// TIA Portal V20 export
FUNCTION_BLOCK "CalculateCam_FeedingRoll"   // FB189, SCL
// stored: Access Published, MemoryReserve 100, SetENOAutomatically false
   VAR_INPUT
      targetCam : TO_Cam;
      excute { ExternalAccessible := 'False'; ExternalVisible := 'False'; ExternalWritable := 'False'} : Bool;
      cpm { ExternalAccessible := 'False'; ExternalVisible := 'False'; ExternalWritable := 'False'} : LReal;
      cellSize { ExternalAccessible := 'False'; ExternalVisible := 'False'; ExternalWritable := 'False'} : LReal;
   END_VAR
   VAR_OUTPUT
      done { ExternalAccessible := 'False'; ExternalVisible := 'False'; ExternalWritable := 'False'} : Bool;
      busy { ExternalAccessible := 'False'; ExternalVisible := 'False'; ExternalWritable := 'False'} : Bool;
      error { ExternalAccessible := 'False'; ExternalVisible := 'False'; ExternalWritable := 'False'} : Bool;
      errorID { ExternalAccessible := 'False'; ExternalVisible := 'False'; ExternalWritable := 'False'} : Word;
   END_VAR
   VAR
      instMCInterpolateCam { ExternalAccessible := 'False'; ExternalVisible := 'False'; ExternalWritable := 'False'} : MC_INTERPOLATECAM;
      statCmd { ExternalAccessible := 'False'; ExternalVisible := 'False'; ExternalWritable := 'False'; S7_SetPoint := 'True'} : DInt;
   END_VAR
   VAR_TEMP
      tempCycleTime : LReal;
      tempFeedingTime : LReal;
      tempT : LReal;
      tempCT : LReal;
      tempDT : LReal;
      tempL : LReal;
      tempR : LReal;
      tempCalPos : Array[1..15] of LReal;
      tempCalVel : Array[1..15] of LReal;
      tempCalAcc : Array[1..15] of LReal;
      tempJerk : Array[1..15] of LReal;
      tempAcc : Array[1..15] of LReal;
      tempVel : Array[1..15] of LReal;
      tempPos : Array[1..15] of LReal;
      tempTime : Array[1..15] of LReal;
      tempX : Array[1..15] of LReal;
      tempA0 : Array[1..50] of LReal;
      tempA1 : Array[1..50] of LReal;
      tempA2 : Array[1..50] of LReal;
      tempA3 : Array[1..50] of LReal;
      tempA4 : Array[1..50] of LReal;
      tempMax : Int;
   END_VAR
   VAR CONSTANT
      CC_IDLE : Int;
      CC_RESET : Int := 1;
      CC_CALCULATE : Int := 2;
      CC_INTERPOLATE : Int := 3;
      CC_DONE : Int := 4;
      CC_ERROR : Int := 99;
      BASIC_TIMEDIVE : LReal := 2.0;
      BASIC_FEEDERDIVE : LReal := 2.0;
      BASIC_ACCPART : Int := 3;
   END_VAR
BEGIN
   IF #instMCInterpolateCam.Error
   THEN
       #statCmd := #CC_ERROR;
       #errorID := #instMCInterpolateCam.ErrorId;
   END_IF;

   IF NOT #excute
   THEN
       #statCmd := #CC_IDLE;
   END_IF;
   REGION State machine
       CASE #statCmd
       OF
           #CC_IDLE:
               #errorID := 16#0;

               IF #excute
               THEN
                   #statCmd := #CC_RESET;
               END_IF;

           #CC_RESET:
               #targetCam.Segment[1].xmin := 0.0;
               #targetCam.Segment[2].xmin := 0.0;
               #targetCam.Segment[3].xmin := 0.0;
               #targetCam.Segment[4].xmin := 0.0;
               #targetCam.Segment[5].xmin := 0.0;
               #targetCam.Segment[6].xmin := 0.0;
               #targetCam.Segment[7].xmin := 0.0;
               #targetCam.Segment[8].xmin := 0.0;
               #targetCam.Segment[9].xmin := 0.0;
               #targetCam.Segment[10].xmin := 0.0;
               #targetCam.Segment[11].xmin := 0.0;
               #targetCam.Segment[12].xmin := 0.0;
               #targetCam.Segment[13].xmin := 0.0;
               #targetCam.Segment[14].xmin := 0.0;
               #targetCam.Segment[15].xmin := 0.0;
               #targetCam.Segment[16].xmin := 0.0;
               #targetCam.Segment[17].xmin := 0.0;
               #targetCam.Segment[18].xmin := 0.0;
               #targetCam.Segment[19].xmin := 0.0;
               #targetCam.Segment[20].xmin := 0.0;
               #targetCam.Segment[21].xmin := 0.0;
               #targetCam.Segment[22].xmin := 0.0;
               #targetCam.Segment[23].xmin := 0.0;
               #targetCam.Segment[24].xmin := 0.0;
               #targetCam.Segment[25].xmin := 0.0;
               #targetCam.Segment[26].xmin := 0.0;
               #targetCam.Segment[27].xmin := 0.0;
               #targetCam.Segment[28].xmin := 0.0;
               #targetCam.Segment[29].xmin := 0.0;
               #targetCam.Segment[30].xmin := 0.0;
               #targetCam.Segment[31].xmin := 0.0;
               #targetCam.Segment[32].xmin := 0.0;
               #targetCam.Segment[33].xmin := 0.0;
               #targetCam.Segment[34].xmin := 0.0;
               #targetCam.Segment[35].xmin := 0.0;
               #targetCam.Segment[36].xmin := 0.0;
               #targetCam.Segment[37].xmin := 0.0;
               #targetCam.Segment[38].xmin := 0.0;
               #targetCam.Segment[39].xmin := 0.0;
               #targetCam.Segment[40].xmin := 0.0;
               #targetCam.Segment[41].xmin := 0.0;
               #targetCam.Segment[42].xmin := 0.0;
               #targetCam.Segment[43].xmin := 0.0;
               #targetCam.Segment[44].xmin := 0.0;
               #targetCam.Segment[45].xmin := 0.0;
               #targetCam.Segment[46].xmin := 0.0;
               #targetCam.Segment[47].xmin := 0.0;
               #targetCam.Segment[48].xmin := 0.0;
               #targetCam.Segment[49].xmin := 0.0;
               #targetCam.Segment[50].xmin := 0.0;

               #targetCam.Segment[1].xmax := 0.0;
               #targetCam.Segment[2].xmax := 0.0;
               #targetCam.Segment[3].xmax := 0.0;
               #targetCam.Segment[4].xmax := 0.0;
               #targetCam.Segment[5].xmax := 0.0;
               #targetCam.Segment[6].xmax := 0.0;
               #targetCam.Segment[7].xmax := 0.0;
               #targetCam.Segment[8].xmax := 0.0;
               #targetCam.Segment[9].xmax := 0.0;
               #targetCam.Segment[10].xmax := 0.0;
               #targetCam.Segment[11].xmax := 0.0;
               #targetCam.Segment[12].xmax := 0.0;
               #targetCam.Segment[13].xmax := 0.0;
               #targetCam.Segment[14].xmax := 0.0;
               #targetCam.Segment[15].xmax := 0.0;
               #targetCam.Segment[16].xmax := 0.0;
               #targetCam.Segment[17].xmax := 0.0;
               #targetCam.Segment[18].xmax := 0.0;
               #targetCam.Segment[19].xmax := 0.0;
               #targetCam.Segment[20].xmax := 0.0;
               #targetCam.Segment[21].xmax := 0.0;
               #targetCam.Segment[22].xmax := 0.0;
               #targetCam.Segment[23].xmax := 0.0;
               #targetCam.Segment[24].xmax := 0.0;
               #targetCam.Segment[25].xmax := 0.0;
               #targetCam.Segment[26].xmax := 0.0;
               #targetCam.Segment[27].xmax := 0.0;
               #targetCam.Segment[28].xmax := 0.0;
               #targetCam.Segment[29].xmax := 0.0;
               #targetCam.Segment[30].xmax := 0.0;
               #targetCam.Segment[31].xmax := 0.0;
               #targetCam.Segment[32].xmax := 0.0;
               #targetCam.Segment[33].xmax := 0.0;
               #targetCam.Segment[34].xmax := 0.0;
               #targetCam.Segment[35].xmax := 0.0;
               #targetCam.Segment[36].xmax := 0.0;
               #targetCam.Segment[37].xmax := 0.0;
               #targetCam.Segment[38].xmax := 0.0;
               #targetCam.Segment[39].xmax := 0.0;
               #targetCam.Segment[40].xmax := 0.0;
               #targetCam.Segment[41].xmax := 0.0;
               #targetCam.Segment[42].xmax := 0.0;
               #targetCam.Segment[43].xmax := 0.0;
               #targetCam.Segment[44].xmax := 0.0;
               #targetCam.Segment[45].xmax := 0.0;
               #targetCam.Segment[46].xmax := 0.0;
               #targetCam.Segment[47].xmax := 0.0;
               #targetCam.Segment[48].xmax := 0.0;
               #targetCam.Segment[49].xmax := 0.0;
               #targetCam.Segment[50].xmax := 0.0;

               #targetCam.Segment[1].a0 := 0.0;
               #targetCam.Segment[2].a0 := 0.0;
               #targetCam.Segment[3].a0 := 0.0;
               #targetCam.Segment[4].a0 := 0.0;
               #targetCam.Segment[5].a0 := 0.0;
               #targetCam.Segment[6].a0 := 0.0;
               #targetCam.Segment[7].a0 := 0.0;
               #targetCam.Segment[8].a0 := 0.0;
               #targetCam.Segment[9].a0 := 0.0;
               #targetCam.Segment[10].a0 := 0.0;
               #targetCam.Segment[11].a0 := 0.0;
               #targetCam.Segment[12].a0 := 0.0;
               #targetCam.Segment[13].a0 := 0.0;
               #targetCam.Segment[14].a0 := 0.0;
               #targetCam.Segment[15].a0 := 0.0;
               #targetCam.Segment[16].a0 := 0.0;
               #targetCam.Segment[17].a0 := 0.0;
               #targetCam.Segment[18].a0 := 0.0;
               #targetCam.Segment[19].a0 := 0.0;
               #targetCam.Segment[20].a0 := 0.0;
               #targetCam.Segment[21].a0 := 0.0;
               #targetCam.Segment[22].a0 := 0.0;
               #targetCam.Segment[23].a0 := 0.0;
               #targetCam.Segment[24].a0 := 0.0;
               #targetCam.Segment[25].a0 := 0.0;
               #targetCam.Segment[26].a0 := 0.0;
               #targetCam.Segment[27].a0 := 0.0;
               #targetCam.Segment[28].a0 := 0.0;
               #targetCam.Segment[29].a0 := 0.0;
               #targetCam.Segment[30].a0 := 0.0;
               #targetCam.Segment[31].a0 := 0.0;
               #targetCam.Segment[32].a0 := 0.0;
               #targetCam.Segment[33].a0 := 0.0;
               #targetCam.Segment[34].a0 := 0.0;
               #targetCam.Segment[35].a0 := 0.0;
               #targetCam.Segment[36].a0 := 0.0;
               #targetCam.Segment[37].a0 := 0.0;
               #targetCam.Segment[38].a0 := 0.0;
               #targetCam.Segment[39].a0 := 0.0;
               #targetCam.Segment[40].a0 := 0.0;
               #targetCam.Segment[41].a0 := 0.0;
               #targetCam.Segment[42].a0 := 0.0;
               #targetCam.Segment[43].a0 := 0.0;
               #targetCam.Segment[44].a0 := 0.0;
               #targetCam.Segment[45].a0 := 0.0;
               #targetCam.Segment[46].a0 := 0.0;
               #targetCam.Segment[47].a0 := 0.0;
               #targetCam.Segment[48].a0 := 0.0;
               #targetCam.Segment[49].a0 := 0.0;
               #targetCam.Segment[50].a0 := 0.0;

               #targetCam.Segment[1].a1 := 0.0;
               #targetCam.Segment[2].a1 := 0.0;
               #targetCam.Segment[3].a1 := 0.0;
               #targetCam.Segment[4].a1 := 0.0;
               #targetCam.Segment[5].a1 := 0.0;
               #targetCam.Segment[6].a1 := 0.0;
               #targetCam.Segment[7].a1 := 0.0;
               #targetCam.Segment[8].a1 := 0.0;
               #targetCam.Segment[9].a1 := 0.0;
               #targetCam.Segment[10].a1 := 0.0;
               #targetCam.Segment[11].a1 := 0.0;
               #targetCam.Segment[12].a1 := 0.0;
               #targetCam.Segment[13].a1 := 0.0;
               #targetCam.Segment[14].a1 := 0.0;
               #targetCam.Segment[15].a1 := 0.0;
               #targetCam.Segment[16].a1 := 0.0;
               #targetCam.Segment[17].a1 := 0.0;
               #targetCam.Segment[18].a1 := 0.0;
               #targetCam.Segment[19].a1 := 0.0;
               #targetCam.Segment[20].a1 := 0.0;
               #targetCam.Segment[21].a1 := 0.0;
               #targetCam.Segment[22].a1 := 0.0;
               #targetCam.Segment[23].a1 := 0.0;
               #targetCam.Segment[24].a1 := 0.0;
               #targetCam.Segment[25].a1 := 0.0;
               #targetCam.Segment[26].a1 := 0.0;
               #targetCam.Segment[27].a1 := 0.0;
               #targetCam.Segment[28].a1 := 0.0;
               #targetCam.Segment[29].a1 := 0.0;
               #targetCam.Segment[30].a1 := 0.0;
               #targetCam.Segment[31].a1 := 0.0;
               #targetCam.Segment[32].a1 := 0.0;
               #targetCam.Segment[33].a1 := 0.0;
               #targetCam.Segment[34].a1 := 0.0;
               #targetCam.Segment[35].a1 := 0.0;
               #targetCam.Segment[36].a1 := 0.0;
               #targetCam.Segment[37].a1 := 0.0;
               #targetCam.Segment[38].a1 := 0.0;
               #targetCam.Segment[39].a1 := 0.0;
               #targetCam.Segment[40].a1 := 0.0;
               #targetCam.Segment[41].a1 := 0.0;
               #targetCam.Segment[42].a1 := 0.0;
               #targetCam.Segment[43].a1 := 0.0;
               #targetCam.Segment[44].a1 := 0.0;
               #targetCam.Segment[45].a1 := 0.0;
               #targetCam.Segment[46].a1 := 0.0;
               #targetCam.Segment[47].a1 := 0.0;
               #targetCam.Segment[48].a1 := 0.0;
               #targetCam.Segment[49].a1 := 0.0;
               #targetCam.Segment[50].a1 := 0.0;

               #targetCam.Segment[1].a2 := 0.0;
               #targetCam.Segment[2].a2 := 0.0;
               #targetCam.Segment[3].a2 := 0.0;
               #targetCam.Segment[4].a2 := 0.0;
               #targetCam.Segment[5].a2 := 0.0;
               #targetCam.Segment[6].a2 := 0.0;
               #targetCam.Segment[7].a2 := 0.0;
               #targetCam.Segment[8].a2 := 0.0;
               #targetCam.Segment[9].a2 := 0.0;
               #targetCam.Segment[10].a2 := 0.0;
               #targetCam.Segment[11].a2 := 0.0;
               #targetCam.Segment[12].a2 := 0.0;
               #targetCam.Segment[13].a2 := 0.0;
               #targetCam.Segment[14].a2 := 0.0;
               #targetCam.Segment[15].a2 := 0.0;
               #targetCam.Segment[16].a2 := 0.0;
               #targetCam.Segment[17].a2 := 0.0;
               #targetCam.Segment[18].a2 := 0.0;
               #targetCam.Segment[19].a2 := 0.0;
               #targetCam.Segment[20].a2 := 0.0;
               #targetCam.Segment[21].a2 := 0.0;
               #targetCam.Segment[22].a2 := 0.0;
               #targetCam.Segment[23].a2 := 0.0;
               #targetCam.Segment[24].a2 := 0.0;
               #targetCam.Segment[25].a2 := 0.0;
               #targetCam.Segment[26].a2 := 0.0;
               #targetCam.Segment[27].a2 := 0.0;
               #targetCam.Segment[28].a2 := 0.0;
               #targetCam.Segment[29].a2 := 0.0;
               #targetCam.Segment[30].a2 := 0.0;
               #targetCam.Segment[31].a2 := 0.0;
               #targetCam.Segment[32].a2 := 0.0;
               #targetCam.Segment[33].a2 := 0.0;
               #targetCam.Segment[34].a2 := 0.0;
               #targetCam.Segment[35].a2 := 0.0;
               #targetCam.Segment[36].a2 := 0.0;
               #targetCam.Segment[37].a2 := 0.0;
               #targetCam.Segment[38].a2 := 0.0;
               #targetCam.Segment[39].a2 := 0.0;
               #targetCam.Segment[40].a2 := 0.0;
               #targetCam.Segment[41].a2 := 0.0;
               #targetCam.Segment[42].a2 := 0.0;
               #targetCam.Segment[43].a2 := 0.0;
               #targetCam.Segment[44].a2 := 0.0;
               #targetCam.Segment[45].a2 := 0.0;
               #targetCam.Segment[46].a2 := 0.0;
               #targetCam.Segment[47].a2 := 0.0;
               #targetCam.Segment[48].a2 := 0.0;
               #targetCam.Segment[49].a2 := 0.0;
               #targetCam.Segment[50].a2 := 0.0;

               #targetCam.Segment[1].a3 := 0.0;
               #targetCam.Segment[2].a3 := 0.0;
               #targetCam.Segment[3].a3 := 0.0;
               #targetCam.Segment[4].a3 := 0.0;
               #targetCam.Segment[5].a3 := 0.0;
               #targetCam.Segment[6].a3 := 0.0;
               #targetCam.Segment[7].a3 := 0.0;
               #targetCam.Segment[8].a3 := 0.0;
               #targetCam.Segment[9].a3 := 0.0;
               #targetCam.Segment[10].a3 := 0.0;
               #targetCam.Segment[11].a3 := 0.0;
               #targetCam.Segment[12].a3 := 0.0;
               #targetCam.Segment[13].a3 := 0.0;
               #targetCam.Segment[14].a3 := 0.0;
               #targetCam.Segment[15].a3 := 0.0;
               #targetCam.Segment[16].a3 := 0.0;
               #targetCam.Segment[17].a3 := 0.0;
               #targetCam.Segment[18].a3 := 0.0;
               #targetCam.Segment[19].a3 := 0.0;
               #targetCam.Segment[20].a3 := 0.0;
               #targetCam.Segment[21].a3 := 0.0;
               #targetCam.Segment[22].a3 := 0.0;
               #targetCam.Segment[23].a3 := 0.0;
               #targetCam.Segment[24].a3 := 0.0;
               #targetCam.Segment[25].a3 := 0.0;
               #targetCam.Segment[26].a3 := 0.0;
               #targetCam.Segment[27].a3 := 0.0;
               #targetCam.Segment[28].a3 := 0.0;
               #targetCam.Segment[29].a3 := 0.0;
               #targetCam.Segment[30].a3 := 0.0;
               #targetCam.Segment[31].a3 := 0.0;
               #targetCam.Segment[32].a3 := 0.0;
               #targetCam.Segment[33].a3 := 0.0;
               #targetCam.Segment[34].a3 := 0.0;
               #targetCam.Segment[35].a3 := 0.0;
               #targetCam.Segment[36].a3 := 0.0;
               #targetCam.Segment[37].a3 := 0.0;
               #targetCam.Segment[38].a3 := 0.0;
               #targetCam.Segment[39].a3 := 0.0;
               #targetCam.Segment[40].a3 := 0.0;
               #targetCam.Segment[41].a3 := 0.0;
               #targetCam.Segment[42].a3 := 0.0;
               #targetCam.Segment[43].a3 := 0.0;
               #targetCam.Segment[44].a3 := 0.0;
               #targetCam.Segment[45].a3 := 0.0;
               #targetCam.Segment[46].a3 := 0.0;
               #targetCam.Segment[47].a3 := 0.0;
               #targetCam.Segment[48].a3 := 0.0;
               #targetCam.Segment[49].a3 := 0.0;
               #targetCam.Segment[50].a3 := 0.0;

               #targetCam.Segment[1].a4 := 0.0;
               #targetCam.Segment[2].a4 := 0.0;
               #targetCam.Segment[3].a4 := 0.0;
               #targetCam.Segment[4].a4 := 0.0;
               #targetCam.Segment[5].a4 := 0.0;
               #targetCam.Segment[6].a4 := 0.0;
               #targetCam.Segment[7].a4 := 0.0;
               #targetCam.Segment[8].a4 := 0.0;
               #targetCam.Segment[9].a4 := 0.0;
               #targetCam.Segment[10].a4 := 0.0;
               #targetCam.Segment[11].a4 := 0.0;
               #targetCam.Segment[12].a4 := 0.0;
               #targetCam.Segment[13].a4 := 0.0;
               #targetCam.Segment[14].a4 := 0.0;
               #targetCam.Segment[15].a4 := 0.0;
               #targetCam.Segment[16].a4 := 0.0;
               #targetCam.Segment[17].a4 := 0.0;
               #targetCam.Segment[18].a4 := 0.0;
               #targetCam.Segment[19].a4 := 0.0;
               #targetCam.Segment[20].a4 := 0.0;
               #targetCam.Segment[21].a4 := 0.0;
               #targetCam.Segment[22].a4 := 0.0;
               #targetCam.Segment[23].a4 := 0.0;
               #targetCam.Segment[24].a4 := 0.0;
               #targetCam.Segment[25].a4 := 0.0;
               #targetCam.Segment[26].a4 := 0.0;
               #targetCam.Segment[27].a4 := 0.0;
               #targetCam.Segment[28].a4 := 0.0;
               #targetCam.Segment[29].a4 := 0.0;
               #targetCam.Segment[30].a4 := 0.0;
               #targetCam.Segment[31].a4 := 0.0;
               #targetCam.Segment[32].a4 := 0.0;
               #targetCam.Segment[33].a4 := 0.0;
               #targetCam.Segment[34].a4 := 0.0;
               #targetCam.Segment[35].a4 := 0.0;
               #targetCam.Segment[36].a4 := 0.0;
               #targetCam.Segment[37].a4 := 0.0;
               #targetCam.Segment[38].a4 := 0.0;
               #targetCam.Segment[39].a4 := 0.0;
               #targetCam.Segment[40].a4 := 0.0;
               #targetCam.Segment[41].a4 := 0.0;
               #targetCam.Segment[42].a4 := 0.0;
               #targetCam.Segment[43].a4 := 0.0;
               #targetCam.Segment[44].a4 := 0.0;
               #targetCam.Segment[45].a4 := 0.0;
               #targetCam.Segment[46].a4 := 0.0;
               #targetCam.Segment[47].a4 := 0.0;
               #targetCam.Segment[48].a4 := 0.0;
               #targetCam.Segment[49].a4 := 0.0;
               #targetCam.Segment[50].a4 := 0.0;

               #targetCam.Segment[1].a5 := 0.0;
               #targetCam.Segment[2].a5 := 0.0;
               #targetCam.Segment[3].a5 := 0.0;
               #targetCam.Segment[4].a5 := 0.0;
               #targetCam.Segment[5].a5 := 0.0;
               #targetCam.Segment[6].a5 := 0.0;
               #targetCam.Segment[7].a5 := 0.0;
               #targetCam.Segment[8].a5 := 0.0;
               #targetCam.Segment[9].a5 := 0.0;
               #targetCam.Segment[10].a5 := 0.0;
               #targetCam.Segment[11].a5 := 0.0;
               #targetCam.Segment[12].a5 := 0.0;
               #targetCam.Segment[13].a5 := 0.0;
               #targetCam.Segment[14].a5 := 0.0;
               #targetCam.Segment[15].a5 := 0.0;
               #targetCam.Segment[16].a5 := 0.0;
               #targetCam.Segment[17].a5 := 0.0;
               #targetCam.Segment[18].a5 := 0.0;
               #targetCam.Segment[19].a5 := 0.0;
               #targetCam.Segment[20].a5 := 0.0;
               #targetCam.Segment[21].a5 := 0.0;
               #targetCam.Segment[22].a5 := 0.0;
               #targetCam.Segment[23].a5 := 0.0;
               #targetCam.Segment[24].a5 := 0.0;
               #targetCam.Segment[25].a5 := 0.0;
               #targetCam.Segment[26].a5 := 0.0;
               #targetCam.Segment[27].a5 := 0.0;
               #targetCam.Segment[28].a5 := 0.0;
               #targetCam.Segment[29].a5 := 0.0;
               #targetCam.Segment[30].a5 := 0.0;
               #targetCam.Segment[31].a5 := 0.0;
               #targetCam.Segment[32].a5 := 0.0;
               #targetCam.Segment[33].a5 := 0.0;
               #targetCam.Segment[34].a5 := 0.0;
               #targetCam.Segment[35].a5 := 0.0;
               #targetCam.Segment[36].a5 := 0.0;
               #targetCam.Segment[37].a5 := 0.0;
               #targetCam.Segment[38].a5 := 0.0;
               #targetCam.Segment[39].a5 := 0.0;
               #targetCam.Segment[40].a5 := 0.0;
               #targetCam.Segment[41].a5 := 0.0;
               #targetCam.Segment[42].a5 := 0.0;
               #targetCam.Segment[43].a5 := 0.0;
               #targetCam.Segment[44].a5 := 0.0;
               #targetCam.Segment[45].a5 := 0.0;
               #targetCam.Segment[46].a5 := 0.0;
               #targetCam.Segment[47].a5 := 0.0;
               #targetCam.Segment[48].a5 := 0.0;
               #targetCam.Segment[49].a5 := 0.0;
               #targetCam.Segment[50].a5 := 0.0;

               #targetCam.Segment[1].a6 := 0.0;
               #targetCam.Segment[2].a6 := 0.0;
               #targetCam.Segment[3].a6 := 0.0;
               #targetCam.Segment[4].a6 := 0.0;
               #targetCam.Segment[5].a6 := 0.0;
               #targetCam.Segment[6].a6 := 0.0;
               #targetCam.Segment[7].a6 := 0.0;
               #targetCam.Segment[8].a6 := 0.0;
               #targetCam.Segment[9].a6 := 0.0;
               #targetCam.Segment[10].a6 := 0.0;
               #targetCam.Segment[11].a6 := 0.0;
               #targetCam.Segment[12].a6 := 0.0;
               #targetCam.Segment[13].a6 := 0.0;
               #targetCam.Segment[14].a6 := 0.0;
               #targetCam.Segment[15].a6 := 0.0;
               #targetCam.Segment[16].a6 := 0.0;
               #targetCam.Segment[17].a6 := 0.0;
               #targetCam.Segment[18].a6 := 0.0;
               #targetCam.Segment[19].a6 := 0.0;
               #targetCam.Segment[20].a6 := 0.0;
               #targetCam.Segment[21].a6 := 0.0;
               #targetCam.Segment[22].a6 := 0.0;
               #targetCam.Segment[23].a6 := 0.0;
               #targetCam.Segment[24].a6 := 0.0;
               #targetCam.Segment[25].a6 := 0.0;
               #targetCam.Segment[26].a6 := 0.0;
               #targetCam.Segment[27].a6 := 0.0;
               #targetCam.Segment[28].a6 := 0.0;
               #targetCam.Segment[29].a6 := 0.0;
               #targetCam.Segment[30].a6 := 0.0;
               #targetCam.Segment[31].a6 := 0.0;
               #targetCam.Segment[32].a6 := 0.0;
               #targetCam.Segment[33].a6 := 0.0;
               #targetCam.Segment[34].a6 := 0.0;
               #targetCam.Segment[35].a6 := 0.0;
               #targetCam.Segment[36].a6 := 0.0;
               #targetCam.Segment[37].a6 := 0.0;
               #targetCam.Segment[38].a6 := 0.0;
               #targetCam.Segment[39].a6 := 0.0;
               #targetCam.Segment[40].a6 := 0.0;
               #targetCam.Segment[41].a6 := 0.0;
               #targetCam.Segment[42].a6 := 0.0;
               #targetCam.Segment[43].a6 := 0.0;
               #targetCam.Segment[44].a6 := 0.0;
               #targetCam.Segment[45].a6 := 0.0;
               #targetCam.Segment[46].a6 := 0.0;
               #targetCam.Segment[47].a6 := 0.0;
               #targetCam.Segment[48].a6 := 0.0;
               #targetCam.Segment[49].a6 := 0.0;
               #targetCam.Segment[50].a6 := 0.0;

               #targetCam.Segment[1].sineAmplitude := 0.0;
               #targetCam.Segment[2].sineAmplitude := 0.0;
               #targetCam.Segment[3].sineAmplitude := 0.0;
               #targetCam.Segment[4].sineAmplitude := 0.0;
               #targetCam.Segment[5].sineAmplitude := 0.0;
               #targetCam.Segment[6].sineAmplitude := 0.0;
               #targetCam.Segment[7].sineAmplitude := 0.0;
               #targetCam.Segment[8].sineAmplitude := 0.0;
               #targetCam.Segment[9].sineAmplitude := 0.0;
               #targetCam.Segment[10].sineAmplitude := 0.0;
               #targetCam.Segment[11].sineAmplitude := 0.0;
               #targetCam.Segment[12].sineAmplitude := 0.0;
               #targetCam.Segment[13].sineAmplitude := 0.0;
               #targetCam.Segment[14].sineAmplitude := 0.0;
               #targetCam.Segment[15].sineAmplitude := 0.0;
               #targetCam.Segment[16].sineAmplitude := 0.0;
               #targetCam.Segment[17].sineAmplitude := 0.0;
               #targetCam.Segment[18].sineAmplitude := 0.0;
               #targetCam.Segment[19].sineAmplitude := 0.0;
               #targetCam.Segment[20].sineAmplitude := 0.0;
               #targetCam.Segment[21].sineAmplitude := 0.0;
               #targetCam.Segment[22].sineAmplitude := 0.0;
               #targetCam.Segment[23].sineAmplitude := 0.0;
               #targetCam.Segment[24].sineAmplitude := 0.0;
               #targetCam.Segment[25].sineAmplitude := 0.0;
               #targetCam.Segment[26].sineAmplitude := 0.0;
               #targetCam.Segment[27].sineAmplitude := 0.0;
               #targetCam.Segment[28].sineAmplitude := 0.0;
               #targetCam.Segment[29].sineAmplitude := 0.0;
               #targetCam.Segment[30].sineAmplitude := 0.0;
               #targetCam.Segment[31].sineAmplitude := 0.0;
               #targetCam.Segment[32].sineAmplitude := 0.0;
               #targetCam.Segment[33].sineAmplitude := 0.0;
               #targetCam.Segment[34].sineAmplitude := 0.0;
               #targetCam.Segment[35].sineAmplitude := 0.0;
               #targetCam.Segment[36].sineAmplitude := 0.0;
               #targetCam.Segment[37].sineAmplitude := 0.0;
               #targetCam.Segment[38].sineAmplitude := 0.0;
               #targetCam.Segment[39].sineAmplitude := 0.0;
               #targetCam.Segment[40].sineAmplitude := 0.0;
               #targetCam.Segment[41].sineAmplitude := 0.0;
               #targetCam.Segment[42].sineAmplitude := 0.0;
               #targetCam.Segment[43].sineAmplitude := 0.0;
               #targetCam.Segment[44].sineAmplitude := 0.0;
               #targetCam.Segment[45].sineAmplitude := 0.0;
               #targetCam.Segment[46].sineAmplitude := 0.0;
               #targetCam.Segment[47].sineAmplitude := 0.0;
               #targetCam.Segment[48].sineAmplitude := 0.0;
               #targetCam.Segment[49].sineAmplitude := 0.0;
               #targetCam.Segment[50].sineAmplitude := 0.0;

               #targetCam.Segment[1].sinePeriod := 0.0;
               #targetCam.Segment[2].sinePeriod := 0.0;
               #targetCam.Segment[3].sinePeriod := 0.0;
               #targetCam.Segment[4].sinePeriod := 0.0;
               #targetCam.Segment[5].sinePeriod := 0.0;
               #targetCam.Segment[6].sinePeriod := 0.0;
               #targetCam.Segment[7].sinePeriod := 0.0;
               #targetCam.Segment[8].sinePeriod := 0.0;
               #targetCam.Segment[9].sinePeriod := 0.0;
               #targetCam.Segment[10].sinePeriod := 0.0;
               #targetCam.Segment[11].sinePeriod := 0.0;
               #targetCam.Segment[12].sinePeriod := 0.0;
               #targetCam.Segment[13].sinePeriod := 0.0;
               #targetCam.Segment[14].sinePeriod := 0.0;
               #targetCam.Segment[15].sinePeriod := 0.0;
               #targetCam.Segment[16].sinePeriod := 0.0;
               #targetCam.Segment[17].sinePeriod := 0.0;
               #targetCam.Segment[18].sinePeriod := 0.0;
               #targetCam.Segment[19].sinePeriod := 0.0;
               #targetCam.Segment[20].sinePeriod := 0.0;
               #targetCam.Segment[21].sinePeriod := 0.0;
               #targetCam.Segment[22].sinePeriod := 0.0;
               #targetCam.Segment[23].sinePeriod := 0.0;
               #targetCam.Segment[24].sinePeriod := 0.0;
               #targetCam.Segment[25].sinePeriod := 0.0;
               #targetCam.Segment[26].sinePeriod := 0.0;
               #targetCam.Segment[27].sinePeriod := 0.0;
               #targetCam.Segment[28].sinePeriod := 0.0;
               #targetCam.Segment[29].sinePeriod := 0.0;
               #targetCam.Segment[30].sinePeriod := 0.0;
               #targetCam.Segment[31].sinePeriod := 0.0;
               #targetCam.Segment[32].sinePeriod := 0.0;
               #targetCam.Segment[33].sinePeriod := 0.0;
               #targetCam.Segment[34].sinePeriod := 0.0;
               #targetCam.Segment[35].sinePeriod := 0.0;
               #targetCam.Segment[36].sinePeriod := 0.0;
               #targetCam.Segment[37].sinePeriod := 0.0;
               #targetCam.Segment[38].sinePeriod := 0.0;
               #targetCam.Segment[39].sinePeriod := 0.0;
               #targetCam.Segment[40].sinePeriod := 0.0;
               #targetCam.Segment[41].sinePeriod := 0.0;
               #targetCam.Segment[42].sinePeriod := 0.0;
               #targetCam.Segment[43].sinePeriod := 0.0;
               #targetCam.Segment[44].sinePeriod := 0.0;
               #targetCam.Segment[45].sinePeriod := 0.0;
               #targetCam.Segment[46].sinePeriod := 0.0;
               #targetCam.Segment[47].sinePeriod := 0.0;
               #targetCam.Segment[48].sinePeriod := 0.0;
               #targetCam.Segment[49].sinePeriod := 0.0;
               #targetCam.Segment[50].sinePeriod := 0.0;

               #targetCam.Segment[1].sinePhase := 0.0;
               #targetCam.Segment[2].sinePhase := 0.0;
               #targetCam.Segment[3].sinePhase := 0.0;
               #targetCam.Segment[4].sinePhase := 0.0;
               #targetCam.Segment[5].sinePhase := 0.0;
               #targetCam.Segment[6].sinePhase := 0.0;
               #targetCam.Segment[7].sinePhase := 0.0;
               #targetCam.Segment[8].sinePhase := 0.0;
               #targetCam.Segment[9].sinePhase := 0.0;
               #targetCam.Segment[10].sinePhase := 0.0;
               #targetCam.Segment[11].sinePhase := 0.0;
               #targetCam.Segment[12].sinePhase := 0.0;
               #targetCam.Segment[13].sinePhase := 0.0;
               #targetCam.Segment[14].sinePhase := 0.0;
               #targetCam.Segment[15].sinePhase := 0.0;
               #targetCam.Segment[16].sinePhase := 0.0;
               #targetCam.Segment[17].sinePhase := 0.0;
               #targetCam.Segment[18].sinePhase := 0.0;
               #targetCam.Segment[19].sinePhase := 0.0;
               #targetCam.Segment[20].sinePhase := 0.0;
               #targetCam.Segment[21].sinePhase := 0.0;
               #targetCam.Segment[22].sinePhase := 0.0;
               #targetCam.Segment[23].sinePhase := 0.0;
               #targetCam.Segment[24].sinePhase := 0.0;
               #targetCam.Segment[25].sinePhase := 0.0;
               #targetCam.Segment[26].sinePhase := 0.0;
               #targetCam.Segment[27].sinePhase := 0.0;
               #targetCam.Segment[28].sinePhase := 0.0;
               #targetCam.Segment[29].sinePhase := 0.0;
               #targetCam.Segment[30].sinePhase := 0.0;
               #targetCam.Segment[31].sinePhase := 0.0;
               #targetCam.Segment[32].sinePhase := 0.0;
               #targetCam.Segment[33].sinePhase := 0.0;
               #targetCam.Segment[34].sinePhase := 0.0;
               #targetCam.Segment[35].sinePhase := 0.0;
               #targetCam.Segment[36].sinePhase := 0.0;
               #targetCam.Segment[37].sinePhase := 0.0;
               #targetCam.Segment[38].sinePhase := 0.0;
               #targetCam.Segment[39].sinePhase := 0.0;
               #targetCam.Segment[40].sinePhase := 0.0;
               #targetCam.Segment[41].sinePhase := 0.0;
               #targetCam.Segment[42].sinePhase := 0.0;
               #targetCam.Segment[43].sinePhase := 0.0;
               #targetCam.Segment[44].sinePhase := 0.0;
               #targetCam.Segment[45].sinePhase := 0.0;
               #targetCam.Segment[46].sinePhase := 0.0;
               #targetCam.Segment[47].sinePhase := 0.0;
               #targetCam.Segment[48].sinePhase := 0.0;
               #targetCam.Segment[49].sinePhase := 0.0;
               #targetCam.Segment[50].sinePhase := 0.0;

               #targetCam.ValidSegment[1] := FALSE;
               #targetCam.ValidSegment[2] := FALSE;
               #targetCam.ValidSegment[3] := FALSE;
               #targetCam.ValidSegment[4] := FALSE;
               #targetCam.ValidSegment[5] := FALSE;
               #targetCam.ValidSegment[6] := FALSE;
               #targetCam.ValidSegment[7] := FALSE;
               #targetCam.ValidSegment[8] := FALSE;
               #targetCam.ValidSegment[9] := FALSE;
               #targetCam.ValidSegment[10] := FALSE;
               #targetCam.ValidSegment[11] := FALSE;
               #targetCam.ValidSegment[12] := FALSE;
               #targetCam.ValidSegment[13] := FALSE;
               #targetCam.ValidSegment[14] := FALSE;
               #targetCam.ValidSegment[15] := FALSE;
               #targetCam.ValidSegment[16] := FALSE;
               #targetCam.ValidSegment[17] := FALSE;
               #targetCam.ValidSegment[18] := FALSE;
               #targetCam.ValidSegment[19] := FALSE;
               #targetCam.ValidSegment[20] := FALSE;
               #targetCam.ValidSegment[21] := FALSE;
               #targetCam.ValidSegment[22] := FALSE;
               #targetCam.ValidSegment[23] := FALSE;
               #targetCam.ValidSegment[24] := FALSE;
               #targetCam.ValidSegment[25] := FALSE;
               #targetCam.ValidSegment[26] := FALSE;
               #targetCam.ValidSegment[27] := FALSE;
               #targetCam.ValidSegment[28] := FALSE;
               #targetCam.ValidSegment[29] := FALSE;
               #targetCam.ValidSegment[30] := FALSE;
               #targetCam.ValidSegment[31] := FALSE;
               #targetCam.ValidSegment[32] := FALSE;
               #targetCam.ValidSegment[33] := FALSE;
               #targetCam.ValidSegment[34] := FALSE;
               #targetCam.ValidSegment[35] := FALSE;
               #targetCam.ValidSegment[36] := FALSE;
               #targetCam.ValidSegment[37] := FALSE;
               #targetCam.ValidSegment[38] := FALSE;
               #targetCam.ValidSegment[39] := FALSE;
               #targetCam.ValidSegment[40] := FALSE;
               #targetCam.ValidSegment[41] := FALSE;
               #targetCam.ValidSegment[42] := FALSE;
               #targetCam.ValidSegment[43] := FALSE;
               #targetCam.ValidSegment[44] := FALSE;
               #targetCam.ValidSegment[45] := FALSE;
               #targetCam.ValidSegment[46] := FALSE;
               #targetCam.ValidSegment[47] := FALSE;
               #targetCam.ValidSegment[48] := FALSE;
               #targetCam.ValidSegment[49] := FALSE;
               #targetCam.ValidSegment[50] := FALSE;

               #statCmd := #CC_CALCULATE;

           #CC_CALCULATE:

               // Calculate Value
               #tempCycleTime := 60000.0 / #cpm;
               // CycleTime Calculate
               #tempFeedingTime := #tempCycleTime / #BASIC_TIMEDIVE;
               #tempT := #tempFeedingTime / 2.0;
               // TimePart Calculate Time / 3
               #tempL := #cpm * #cellSize / 60.0;
               #tempR := #cellSize / #tempT * 1000.0;
               // VelocityPart Calculate
               // 
               #tempTime[1] := 0.0;
               #tempTime[2] := #tempL * #tempT / 1000.0;
               #tempTime[3] := #tempL * #tempT / 1000.0;
               #tempTime[4] := 0.0;
               // Calculate Time

               #tempPos[1] := 0.0;
               #tempPos[2] := #tempR * #tempT / 1000.0 / 2.0;
               #tempPos[3] := #tempR * #tempT / 1000.0 / 2.0;
               #tempPos[4] := 0.0;
               // Calculate Pos

               #tempVel[1] := 0.0;
               #tempVel[2] := 2.0 * #tempPos[2] / #tempTime[2];
               #tempVel[3] := 2.0 * #tempPos[3] / #tempTime[3];
               #tempVel[4] := 0.0;

               // Calculate New Vel

               #tempAcc[1] := 0.0;
               #tempAcc[2] := 2.0 * #tempVel[2] / #tempTime[2];
               #tempAcc[3] := - 2.0 * #tempVel[3] / #tempTime[3];
               #tempAcc[4] := 0.0;
               // Calculate Accelation

               #tempJerk[1] := 0.0;
               #tempJerk[2] := 2.0 * #tempAcc[2] / #tempTime[2];
               #tempJerk[3] := - 2.0 * #tempAcc[2] / #tempTime[2];
               #tempJerk[4] := 2.0 * #tempAcc[3] / #tempTime[3];
               #tempJerk[5] := - 2.0 * #tempAcc[3] / #tempTime[3];
               #tempJerk[6] := 0.0;

               // Calculate Jounce

               #tempX[1] := #tempTime[1];
               #tempX[2] := #tempTime[2] / 2.0;
               #tempX[3] := #tempTime[2] / 2.0;
               #tempX[4] := #tempTime[3] / 2.0;
               #tempX[5] := #tempTime[3] / 2.0;
               #tempX[6] := #tempTime[4];

               // Calculate X

               #tempCalAcc[1] := 0.0;
               #tempCalVel[1] := 0.0;
               #tempCalPos[1] := 0.0;
               #tempA3[1] := #tempJerk[1] / 6.0;
               #tempA2[1] := #tempCalAcc[1] / 2.0;
               #tempA1[1] := #tempCalVel[1];
               #tempA0[1] := #tempCalPos[1];
               #targetCam.Segment[1].a0 := #tempA0[1];
               #targetCam.Segment[1].a1 := #tempA1[1];
               #targetCam.Segment[1].a2 := #tempA2[1];
               #targetCam.Segment[1].a3 := #tempA3[1];
               #targetCam.Segment[1].a4 := 0.0;
               #targetCam.Segment[1].a5 := 0.0;
               #targetCam.Segment[1].a6 := 0.0;
               #targetCam.Segment[1].xmax := #tempX[1];
               #targetCam.Segment[1].xmin := 0.0;
               #targetCam.Segment[1].sineAmplitude := 0.0;
               #targetCam.Segment[1].sinePeriod := 0.0;
               #targetCam.Segment[1].sinePhase := 0.0;
               IF #tempX[1] = 0.0 THEN
                   #targetCam.ValidSegment[1] := FALSE;
               ELSE
                   #targetCam.ValidSegment[1] := TRUE;
               END_IF;

               #tempCalAcc[2] := #tempJerk[2 - 1] * #tempX[2 - 1] + #tempCalAcc[2 - 1];
               #tempCalVel[2] := #tempJerk[2 - 1] * #tempX[2 - 1] * #tempX[2 - 1] / 2.0 + #tempCalAcc[2 - 1] * #tempX[2 - 1] + #tempCalVel[2 - 1];
               #tempCalPos[2] := #tempJerk[2 - 1] * #tempX[2 - 1] * #tempX[2 - 1] * #tempX[2 - 1] / 6.0 + #tempCalAcc[2 - 1] * #tempX[2 - 1] * #tempX[2 - 1] / 2.0 + #tempCalVel[2 - 1] * #tempX[2 - 1] + #tempCalPos[2 - 1];
               IF ABS_LREAL(#tempCalVel[2]) < 0.000000001 THEN
                   #tempCalVel[2] := 0.0;
               END_IF;
               IF ABS_LREAL(#tempCalPos[2]) < 0.000000001 THEN
                   #tempCalPos[2] := 0.0;
               END_IF;

               #tempA3[2] := #tempJerk[2] / 6.0;
               #tempA2[2] := #tempCalAcc[2] / 2.0;
               #tempA1[2] := #tempCalVel[2];
               #tempA0[2] := #tempCalPos[2];
               #targetCam.Segment[2].a0 := #tempA0[2];
               #targetCam.Segment[2].a1 := #tempA1[2];
               #targetCam.Segment[2].a2 := #tempA2[2];
               #targetCam.Segment[2].a3 := #tempA3[2];
               #targetCam.Segment[2].a4 := 0.0;
               #targetCam.Segment[2].a5 := 0.0;
               #targetCam.Segment[2].a6 := 0.0;
               #targetCam.Segment[2].xmax := #targetCam.Segment[2 - 1].xmax + #tempX[2];
               #targetCam.Segment[2].xmin := #targetCam.Segment[2 - 1].xmax;
               #targetCam.Segment[2].sineAmplitude := 0.0;
               #targetCam.Segment[2].sinePeriod := 0.0;
               #targetCam.Segment[2].sinePhase := 0.0;
               IF #tempX[2] = 0.0 THEN
                   #targetCam.ValidSegment[2] := FALSE;
               ELSE
                   #targetCam.ValidSegment[2] := TRUE;
               END_IF;

               #tempCalAcc[3] := #tempJerk[3 - 1] * #tempX[3 - 1] + #tempCalAcc[3 - 1];
               #tempCalVel[3] := #tempJerk[3 - 1] * #tempX[3 - 1] * #tempX[3 - 1] / 2.0 + #tempCalAcc[3 - 1] * #tempX[3 - 1] + #tempCalVel[3 - 1];
               #tempCalPos[3] := #tempJerk[3 - 1] * #tempX[3 - 1] * #tempX[3 - 1] * #tempX[3 - 1] / 6.0 + #tempCalAcc[3 - 1] * #tempX[3 - 1] * #tempX[3 - 1] / 2.0 + #tempCalVel[3 - 1] * #tempX[3 - 1] + #tempCalPos[3 - 1];
               IF ABS_LREAL(#tempCalVel[3]) < 0.000000001 THEN
                   #tempCalVel[3] := 0.0;
               END_IF;
               IF ABS_LREAL(#tempCalPos[3]) < 0.000000001 THEN
                   #tempCalPos[3] := 0.0;
               END_IF;

               #tempA3[3] := #tempJerk[3] / 6.0;
               #tempA2[3] := #tempCalAcc[3] / 2.0;
               #tempA1[3] := #tempCalVel[3];
               #tempA0[3] := #tempCalPos[3];
               #targetCam.Segment[3].a0 := #tempA0[3];
               #targetCam.Segment[3].a1 := #tempA1[3];
               #targetCam.Segment[3].a2 := #tempA2[3];
               #targetCam.Segment[3].a3 := #tempA3[3];
               #targetCam.Segment[3].a4 := 0.0;
               #targetCam.Segment[3].a5 := 0.0;
               #targetCam.Segment[3].a6 := 0.0;
               #targetCam.Segment[3].xmax := #targetCam.Segment[3 - 1].xmax + #tempX[3];
               #targetCam.Segment[3].xmin := #targetCam.Segment[3 - 1].xmax;
               #targetCam.Segment[3].sineAmplitude := 0.0;
               #targetCam.Segment[3].sinePeriod := 0.0;
               #targetCam.Segment[3].sinePhase := 0.0;
               IF #tempX[3] = 0.0 THEN
                   #targetCam.ValidSegment[3] := FALSE;
               ELSE
                   #targetCam.ValidSegment[3] := TRUE;
               END_IF;

               #tempCalAcc[4] := #tempJerk[4 - 1] * #tempX[4 - 1] + #tempCalAcc[4 - 1];
               #tempCalVel[4] := #tempJerk[4 - 1] * #tempX[4 - 1] * #tempX[4 - 1] / 2.0 + #tempCalAcc[4 - 1] * #tempX[4 - 1] + #tempCalVel[4 - 1];
               #tempCalPos[4] := #tempJerk[4 - 1] * #tempX[4 - 1] * #tempX[4 - 1] * #tempX[4 - 1] / 6.0 + #tempCalAcc[4 - 1] * #tempX[4 - 1] * #tempX[4 - 1] / 2.0 + #tempCalVel[4 - 1] * #tempX[4 - 1] + #tempCalPos[4 - 1];
               IF ABS_LREAL(#tempCalVel[4]) < 0.000000001 THEN
                   #tempCalVel[4] := 0.0;
               END_IF;
               IF ABS_LREAL(#tempCalPos[4]) < 0.000000001 THEN
                   #tempCalPos[4] := 0.0;
               END_IF;

               #tempA3[4] := #tempJerk[4] / 6.0;
               #tempA2[4] := #tempCalAcc[4] / 2.0;
               #tempA1[4] := #tempCalVel[4];
               #tempA0[4] := #tempCalPos[4];
               #targetCam.Segment[4].a0 := #tempA0[4];
               #targetCam.Segment[4].a1 := #tempA1[4];
               #targetCam.Segment[4].a2 := #tempA2[4];
               #targetCam.Segment[4].a3 := #tempA3[4];
               #targetCam.Segment[4].a4 := 0.0;
               #targetCam.Segment[4].a5 := 0.0;
               #targetCam.Segment[4].a6 := 0.0;
               #targetCam.Segment[4].xmax := #targetCam.Segment[4 - 1].xmax + #tempX[4];
               #targetCam.Segment[4].xmin := #targetCam.Segment[4 - 1].xmax;
               #targetCam.Segment[4].sineAmplitude := 0.0;
               #targetCam.Segment[4].sinePeriod := 0.0;
               #targetCam.Segment[4].sinePhase := 0.0;
               IF #tempX[4] = 0.0 THEN
                   #targetCam.ValidSegment[4] := FALSE;
               ELSE
                   #targetCam.ValidSegment[4] := TRUE;
               END_IF;

               #tempCalAcc[5] := #tempJerk[5 - 1] * #tempX[5 - 1] + #tempCalAcc[5 - 1];
               #tempCalVel[5] := #tempJerk[5 - 1] * #tempX[5 - 1] * #tempX[5 - 1] / 2.0 + #tempCalAcc[5 - 1] * #tempX[5 - 1] + #tempCalVel[5 - 1];
               #tempCalPos[5] := #tempJerk[5 - 1] * #tempX[5 - 1] * #tempX[5 - 1] * #tempX[5 - 1] / 6.0 + #tempCalAcc[5 - 1] * #tempX[5 - 1] * #tempX[5 - 1] / 2.0 + #tempCalVel[5 - 1] * #tempX[5 - 1] + #tempCalPos[5 - 1];
               IF ABS_LREAL(#tempCalVel[5]) < 0.000000001 THEN
                   #tempCalVel[5] := 0.0;
               END_IF;
               IF ABS_LREAL(#tempCalPos[5]) < 0.000000001 THEN
                   #tempCalPos[5] := 0.0;
               END_IF;

               #tempA3[5] := #tempJerk[5] / 6.0;
               #tempA2[5] := #tempCalAcc[5] / 2.0;
               #tempA1[5] := #tempCalVel[5];
               #tempA0[5] := #tempCalPos[5];
               #targetCam.Segment[5].a0 := #tempA0[5];
               #targetCam.Segment[5].a1 := #tempA1[5];
               #targetCam.Segment[5].a2 := #tempA2[5];
               #targetCam.Segment[5].a3 := #tempA3[5];
               #targetCam.Segment[5].a4 := 0.0;
               #targetCam.Segment[5].a5 := 0.0;
               #targetCam.Segment[5].a6 := 0.0;
               #targetCam.Segment[5].xmax := #targetCam.Segment[5 - 1].xmax + #tempX[5];
               #targetCam.Segment[5].xmin := #targetCam.Segment[5 - 1].xmax;
               #targetCam.Segment[5].sineAmplitude := 0.0;
               #targetCam.Segment[5].sinePeriod := 0.0;
               #targetCam.Segment[5].sinePhase := 0.0;
               IF #tempX[5] = 0.0 THEN
                   #targetCam.ValidSegment[5] := FALSE;
               ELSE
                   #targetCam.ValidSegment[5] := TRUE;
               END_IF;

               #tempCalAcc[6] := #tempJerk[6 - 1] * #tempX[6 - 1] + #tempCalAcc[6 - 1];
               #tempCalVel[6] := #tempJerk[6 - 1] * #tempX[6 - 1] * #tempX[6 - 1] / 2.0 + #tempCalAcc[6 - 1] * #tempX[6 - 1] + #tempCalVel[6 - 1];
               #tempCalPos[6] := #tempJerk[6 - 1] * #tempX[6 - 1] * #tempX[6 - 1] * #tempX[6 - 1] / 6.0 + #tempCalAcc[6 - 1] * #tempX[6 - 1] * #tempX[6 - 1] / 2.0 + #tempCalVel[6 - 1] * #tempX[6 - 1] + #tempCalPos[6 - 1];
               IF ABS_LREAL(#tempCalVel[6]) < 0.000000001 THEN
                   #tempCalVel[6] := 0.0;
               END_IF;
               IF ABS_LREAL(#tempCalPos[6]) < 0.000000001 THEN
                   #tempCalPos[6] := 0.0;
               END_IF;

               #tempA3[6] := #tempJerk[6] / 6.0;
               #tempA2[6] := #tempCalAcc[6] / 2.0;
               #tempA1[6] := #tempCalVel[6];
               #tempA0[6] := #tempCalPos[6];
               #targetCam.Segment[6].a0 := #tempA0[6];
               #targetCam.Segment[6].a1 := #tempA1[6];
               #targetCam.Segment[6].a2 := #tempA2[6];
               #targetCam.Segment[6].a3 := #tempA3[6];
               #targetCam.Segment[6].a4 := 0.0;
               #targetCam.Segment[6].a5 := 0.0;
               #targetCam.Segment[6].a6 := 0.0;
               #targetCam.Segment[6].xmax := #targetCam.Segment[6 - 1].xmax + #tempX[6];
               #targetCam.Segment[6].xmin := #targetCam.Segment[6 - 1].xmax;
               #targetCam.Segment[6].sineAmplitude := 0.0;
               #targetCam.Segment[6].sinePeriod := 0.0;
               #targetCam.Segment[6].sinePhase := 0.0;
               IF #tempX[6] = 0.0 THEN
                   #targetCam.ValidSegment[6] := FALSE;
               ELSE
                   #targetCam.ValidSegment[6] := TRUE;
               END_IF;

               #statCmd := #CC_INTERPOLATE;

           #CC_INTERPOLATE:
               IF #instMCInterpolateCam.Done
               THEN
                   #statCmd := #CC_DONE;
               END_IF;

           #CC_DONE:
               ;

           #CC_ERROR:
               ;
       END_CASE;

   END_REGION

   REGION Instances
       #instMCInterpolateCam(Cam := #targetCam,
                             Execute := #statCmd = #CC_INTERPOLATE);
   END_REGION

   REGION Outputs
       #busy := #statCmd = #CC_RESET OR #statCmd = #CC_CALCULATE OR #statCmd = #CC_INTERPOLATE;
       #error := #statCmd = #CC_ERROR;
       #done := #statCmd = #CC_DONE;
   END_REGION
END_FUNCTION_BLOCK
